{attribute 'qualified_only'}
VAR_GLOBAL CONSTANT
	nMaxMsgCount : UINT := 10;
	
	nCmd_Mask : UINT := 2#11_1110_0000;
	nCmd_Shift : UINT := 5;
	nNodeId_Mask : UINT := 2#1111_1100_0000_0000;
	nNodeId_Shift : UINT := 10;
	
	nReceiveData_TimeOut : TIME := T#1S;
END_VAR

(* stored: Version 1.1.0.1
   GVL GVL_ODrive: Id {cb6373c8-784a-4720-8009-b8b0b32c3a8b} *)
